// TIA Portal V16 export
// export: Created 2021-03-05T14:22:13.1773459Z, ExportSetting WithDefaults, DisplayName Totally Integrated Automation Portal, DisplayVersion V16, DisplayName TIA Portal Version Control Interface, DisplayVersion V16, DisplayName TIA Portal Openness, DisplayVersion V16, DisplayName SINAMICS Startdrive Advanced, DisplayVersion V16, DisplayName SINAMICS Startdrive G130, G150, S120, S150, SINAMICS MV, S210, DisplayVersion V16, DisplayName SINAMICS Startdrive G110M, G120, G120C, G120D, G120P, DisplayVersion V16, DisplayName STEP 7 Professional, DisplayVersion V16, DisplayName STEP 7 Safety, DisplayVersion V16, DisplayName WinCC Professional, DisplayVersion V16
DATA_BLOCK "dbMain"   // DB5
VERSION : 0.1
// stored: AutoNumber true, DBAccessibleFromOPCUA true, InstanceOfName fbMain, InstanceOfType FB
"fbMain"
   // VAR
   //    Room { ExternalVisible := 'False'} : Array[1.."MAX_ROOMS"] of "fbRoom";
   //    Config { S7_SetPoint := 'True'} : "fbConfig";
   // END_VAR
BEGIN
   Room[1].Rack[3].Fertigation.AI_Reservoir_Level.rHighCalibration := 0.0;
   Room[1].Rack[1].Fertigation.ShelvesFertigation[1].Controls.Flood_Duration := 1;
END_DATA_BLOCK
